TYPE ST_RECORD :
STRUCT
	nID 			: ULINT;
	dtTimeStamp		: DATE_AND_TIME;
	nCustomerID		: DINT;
	nFilmID			: DINT;
END_STRUCT
END_TYPE

(* stored: Version 1.1.0.1
   DUT ST_RECORD: Id {873580b0-4dac-43c6-8c03-b9be14260be0} *)
